(* CODESYS project io.library
   Company: MyCompany
   DefaultNamespace: IO
   Version: 0.1.0.0
   Placeholder: Inputs and Outputs
   Author: Sajedeh Taheri
   Description: this library hold functionality for sensors and actuators
   Title: Inputs and Outputs

Project tree, tasks and I/O mapping:
  libraries: Tc2_Standard, * (Beckhoff Automation GmbH); Tc2_System, * (Beckhoff Automation GmbH); Tc3_Module, * (Beckhoff Automation GmbH)
  DUTs/
  GVLs/
  POUs/
    function F_factorial [ST]
  Version/
    global variables Global_Version
  VISUs/
*)

// Version/Global_Version
{attribute 'TcGenerated'}
{attribute 'no-analysis'}
{attribute 'linkalways'}
// This function has been automatically generated from the project information.
VAR_GLOBAL CONSTANT
	{attribute 'const_non_replaced'}
	stLibVersion_Inputs_and_Outputs : ST_LibVersion := (iMajor := 0, iMinor := 1, iBuild := 0, iRevision := 0, nFlags := 0, sVersion := '0.1.0.0');
END_VAR

// POUs/F_factorial
FUNCTION F_factorial : ULINT
VAR_INPUT
	n : ULINT;
END_VAR
VAR
	tempFact : ULINT;
	i : ULINT;
END_VAR

tempFact := 1;
FOR i := 1 TO n BY 1 DO
	tempFact := i * tempFact;
END_FOR
F_factorial := tempFact;

END_FUNCTION
